Fanuc KAREL source: SET_TPE_CMT.kl

PROGRAM T
%NOLOCKGROUP
VAR
 v0 : INTEGER
 v1 : INTEGER
 v2 : STRING[40]
 v3 : INTEGER
BEGIN
 SET_TPE_CMT(v0, v1, v2, v3)
END T
